// Mitsubishi GX Works2 project: IELET2103_Dataoving_1   PLC: FX2N/FX2NC
// IELET2103_Dataoving_1

// task Task_01 (event TRUE, interval 0, priority 31): Oppgave1

PROGRAM Oppgave1
(* structured ladder/FBD written out as ST: instructions are called as NAME(EN, inputs, outputs); _pN, _eN, _tN stand for wires *)
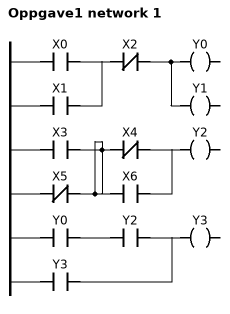
(* network 1 *)
_p1 := (X0 OR X1) AND NOT X2;
Y0 := _p1;
Y1 := _p1;
_p2 := X3 OR (NOT X5);
Y2 := (_p2 AND NOT X4) OR (_p2 AND X6);
Y3 := (Y0 AND Y2) OR Y3;
END_PROGRAM
